(* Schneider Machine Expert - Basic project P1_Part2_PLC+Vulnerabilities, file version 1.6.0.0 *)
(* ProjectInformations: Name=New project *)

HARDWARE
  Cpu 0: TM221M16R/G
  EthernetConfiguration: NetworkName=M221, IpAllocationMode=FixedAddress, IpAddress=0.0.0.0, SubnetMask=0.0.0.0
  SerialLineConfiguration: Baud=Baud19200, Parity=ParityEven, DataBits=DataBits8, StopBits=StopBits1, PhysicalMedium=PhysicalMediumRs485, TransmissionMode=TransmissionModeModbusRtu, SlaveId=1, Addressing=SlaveAddressing
  MastTask: UsePeriodScanMode=false, PeriodScan=100
  FastTask: Period=255
  CpuBehavior: StartingMode=StartAsPreviousState, AutoSaveRamOnEeprom=true, WatchdogPeriod=250

SYMBOLS  (address, symbol, comment, settings)
  %MW0      CURRENT_PRESSURE
  %KW0      PRESSURE_CHECKPOINT  [Value=500]
  %KW1      PRESSURE_CHECKPOINT_UNREACHABLE  [Value=1001]
  %TM0        [Preset=5, Base=OneSecond]
  %I0.0     SHUTDOWN
  %I0.1     CANCEL_SHUTDOWN
  %I0.2     CONFIRM_PRESSURE_CHANGE
  %I0.3     CONFIRM_SHUTDOWN
  %I0.4     EMERGENCY_SHUTDOWN
  %Q0.0     SHUTDOWN_CHECK_1
  %Q0.1     SHUTDOWN_CANCELED
  %Q0.2     SHUTDOWN_CHECK_2
  %Q0.3     SHUTDOWN_CHECK_3
  %Q0.4     EMERGENCY_SHUTDOWN_DECLARED
  %Q0.5     SHUTDOWN_COMPLETED
  %IW0.0    SET_PRESSURE  [Type=Type_0_10V, Scope=Scope_Normal, Minimum=0, Maximum=1000]

POU New POU
  (* SectionNumber=1 *)

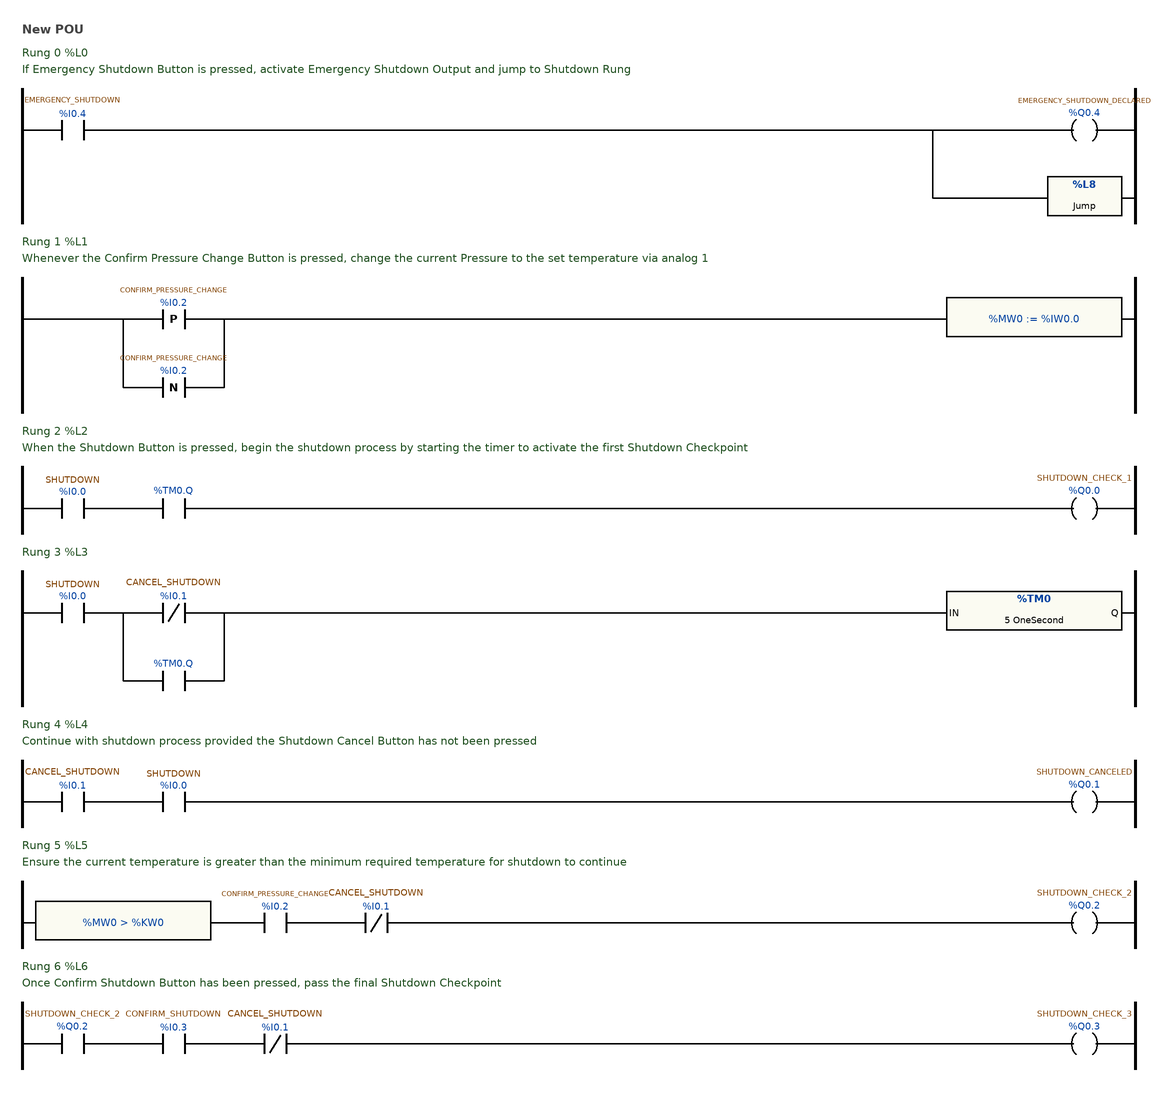

// Rung 0 %L0
// If Emergency Shutdown Button is pressed, activate Emergency Shutdown Output and jump to Shutdown Rung
  %L0:
  LD %I0.4                (* EMERGENCY_SHUTDOWN *)
  ST %Q0.4                (* EMERGENCY_SHUTDOWN_DECLARED *)
  JMPC %L8
  // as ST:
  //   %L0:
  //   EMERGENCY_SHUTDOWN_DECLARED := EMERGENCY_SHUTDOWN;
  //   IF EMERGENCY_SHUTDOWN THEN JMP %L8; END_IF;

// Rung 1 %L1
// Whenever the Confirm Pressure Change Button is pressed, change the current Pressure to the set temperature via analog 1
  %L1:
  LDR %I0.2               (* CONFIRM_PRESSURE_CHANGE *)
  ORF %I0.2               (* CONFIRM_PRESSURE_CHANGE *)
  [ %MW0 := %IW0.0 ]      (* CURRENT_PRESSURE, SET_PRESSURE *)
  // as ST:
  //   %L1:
  //   IF RISING(CONFIRM_PRESSURE_CHANGE) OR FALLING(CONFIRM_PRESSURE_CHANGE) THEN CURRENT_PRESSURE := SET_PRESSURE; END_IF;

// Rung 2 %L2
// When the Shutdown Button is pressed, begin the shutdown process by starting the timer to activate the first Shutdown Checkpoint
  %L2:
  LD %I0.0                (* SHUTDOWN *)
  AND %TM0.Q
  ST %Q0.0                (* SHUTDOWN_CHECK_1 *)
  // as ST:
  //   %L2:
  //   SHUTDOWN_CHECK_1 := SHUTDOWN AND %TM0.Q;

// Rung 3 %L3
  %L3:
  BLK %TM0
  LD %I0.0                (* SHUTDOWN *)
  AND(N %I0.1             (* CANCEL_SHUTDOWN *)
  OR %TM0.Q
  )
  IN
  END_BLK
  // as ST:
  //   %L3:
  //   %TM0(IN := SHUTDOWN AND (NOT CANCEL_SHUTDOWN OR %TM0.Q));

// Rung 4 %L4
// Continue with shutdown process provided the Shutdown Cancel Button has not been pressed
  %L4:
  LD %I0.1                (* CANCEL_SHUTDOWN *)
  AND %I0.0               (* SHUTDOWN *)
  ST %Q0.1                (* SHUTDOWN_CANCELED *)
  // as ST:
  //   %L4:
  //   SHUTDOWN_CANCELED := CANCEL_SHUTDOWN AND SHUTDOWN;

// Rung 5 %L5
// Ensure the current temperature is greater than the minimum required temperature for shutdown to continue
  %L5:
  LD [ %MW0 > %KW0 ]      (* CURRENT_PRESSURE, PRESSURE_CHECKPOINT *)
  AND %I0.2               (* CONFIRM_PRESSURE_CHANGE *)
  ANDN %I0.1              (* CANCEL_SHUTDOWN *)
  ST %Q0.2                (* SHUTDOWN_CHECK_2 *)
  // as ST:
  //   %L5:
  //   SHUTDOWN_CHECK_2 := CURRENT_PRESSURE > PRESSURE_CHECKPOINT AND CONFIRM_PRESSURE_CHANGE AND NOT CANCEL_SHUTDOWN;

// Rung 6 %L6
// Once Confirm Shutdown Button has been pressed, pass the final Shutdown Checkpoint
  %L6:
  LD %Q0.2                (* SHUTDOWN_CHECK_2 *)
  AND %I0.3               (* CONFIRM_SHUTDOWN *)
  ANDN %I0.1              (* CANCEL_SHUTDOWN *)
  ST %Q0.3                (* SHUTDOWN_CHECK_3 *)
  // as ST:
  //   %L6:
  //   SHUTDOWN_CHECK_3 := SHUTDOWN_CHECK_2 AND CONFIRM_SHUTDOWN AND NOT CANCEL_SHUTDOWN;

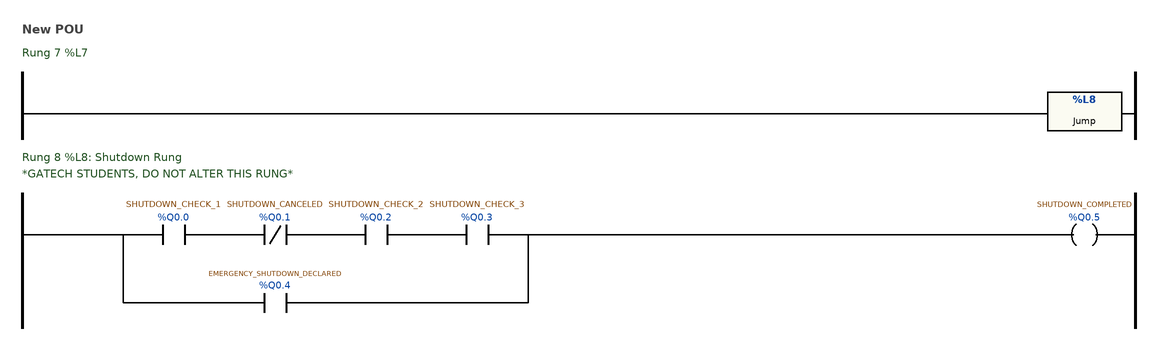

// Rung 7 %L7
  %L7:
  LD 1
  JMPC %L8
  // as ST:
  //   %L7:
  //   JMP %L8;

// Rung 8 %L8: Shutdown Rung
// *GATECH STUDENTS, DO NOT ALTER THIS RUNG*
  %L8:
  LD %Q0.0                (* SHUTDOWN_CHECK_1 *)
  ANDN %Q0.1              (* SHUTDOWN_CANCELED *)
  AND %Q0.2               (* SHUTDOWN_CHECK_2 *)
  AND %Q0.3               (* SHUTDOWN_CHECK_3 *)
  OR %Q0.4                (* EMERGENCY_SHUTDOWN_DECLARED *)
  ST %Q0.5                (* SHUTDOWN_COMPLETED *)
  // as ST:
  //   %L8:
  //   SHUTDOWN_COMPLETED := SHUTDOWN_CHECK_1 AND NOT SHUTDOWN_CANCELED AND SHUTDOWN_CHECK_2 AND SHUTDOWN_CHECK_3 OR EMERGENCY_SHUTDOWN_DECLARED;
